TYPE Modus_Abtauen :
(
		NichtAusgewahlt,
		Abtauen_elektrisch,
		Abtauen_Heissgas_oben,
		Abtauen_Heissgas_unten
);
END_TYPE

(* stored: Version 1.1.0.1, ProductVersion 3.1.4019.2
   DUT Modus_Abtauen: Id {cfb136ed-0116-4be7-b393-79e392ec61b6} *)
